(* Schneider Machine Expert - Basic project resolucao, file version 2.7.0.0 *)
(* ProjectInformations: Name=Novo projeto *)

HARDWARE
  Cpu 0: TM221CE24R
  EthernetConfiguration: NetworkName=M221, IpAllocationMode=FixedAddress, IpAddress=0.0.0.0, SubnetMask=0.0.0.0
  SerialLineConfiguration: Baud=Baud19200, Parity=ParityEven, DataBits=DataBits8, StopBits=StopBits1, PhysicalMedium=PhysicalMediumRs485, TransmissionMode=TransmissionModeModbusRtu, SlaveId=1, Addressing=SlaveAddressing
  MastTask: UsePeriodScanMode=false, PeriodScan=100
  FastTask: Period=255
  CpuBehavior: StartingMode=StartAsPreviousState, AutoSaveRamOnEeprom=true, WatchdogPeriod=250

SYMBOLS  (address, symbol, comment, settings)
  %M0       SIG_LED_1
  %M1       SIG_TM_1
  %M10      SIG_OUT_LED_1
  %TM0      TM_1  [Preset=2, Base=OneSecond]
  %Q0.1     OUT_LED_1

POU Lógicas
  (* SectionNumber=1 *)

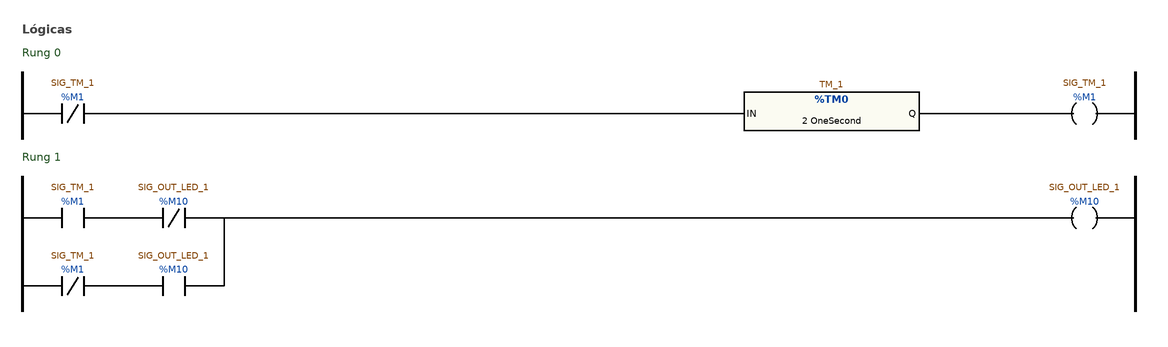

// Rung 0
  BLK %TM0                (* TM_1 *)
  LDN %M1                 (* SIG_TM_1 *)
  IN
  OUT_BLK
  LD Q
  ST %M1                  (* SIG_TM_1 *)
  END_BLK
  // as ST:
  //   TM_1(IN := NOT SIG_TM_1);
  //   SIG_TM_1 := TM_1.Q;

// Rung 1
  LD %M1                  (* SIG_TM_1 *)
  ANDN %M10               (* SIG_OUT_LED_1 *)
  OR(N %M1                (* SIG_TM_1 *)
  AND %M10                (* SIG_OUT_LED_1 *)
  )
  ST %M10                 (* SIG_OUT_LED_1 *)
  // as ST:
  //   SIG_OUT_LED_1 := SIG_TM_1 AND NOT SIG_OUT_LED_1 OR NOT SIG_TM_1 AND SIG_OUT_LED_1;

POU Saídas
  (* SectionNumber=2 *)

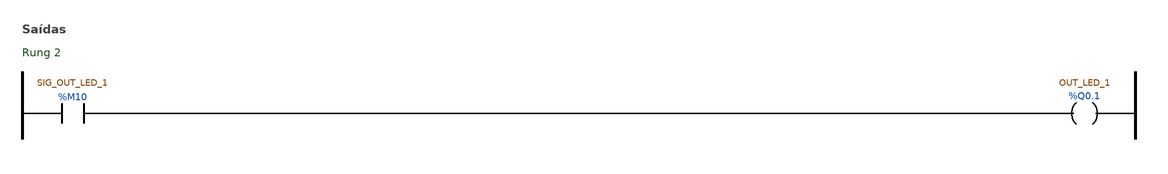

// Rung 2
  LD %M10                 (* SIG_OUT_LED_1 *)
  ST %Q0.1                (* OUT_LED_1 *)
  // as ST:
  //   OUT_LED_1 := SIG_OUT_LED_1;
